PROGRAM POU2
VAR
	puvar2: INT;
END_VAR

puvar2:=4;

END_PROGRAM

(* stored: Version 1.1.0.1, ProductVersion 3.1.4024.9
   POU POU2: Id {31cd0aa8-f9b4-4005-a800-b94a0936a0ec}, SpecialFunc None *)
